(* CODESYS project Library01.library
   Company: MyCompany
   DefaultNamespace: MyNamespace01
   Version: 2.0.0.0
   Placeholder: MyLibrary01
   Title: MyLibrary01

Project tree, tasks and I/O mapping:
  libraries: Tc2_Standard, * (Beckhoff Automation GmbH); Tc2_System, * (Beckhoff Automation GmbH); Tc3_Module, * (Beckhoff Automation GmbH)
  DUTs/
    data type E_Foo
    data type ST_Foo
  GVLs/
    global variables GVL01
  POUs/
    function block FB_Foo [ST]
    interface I_Foo: DoSomething
  Version/
    global variables Global_Version
  VISUs/
*)

// DUTs/E_Foo
// {attribute 'qualified_only'}
// {attribute 'strict'}
TYPE E_Foo :
(
	eRed := 0,
	eBlue := 1,
	eGreen := 2
);
END_TYPE

// DUTs/ST_Foo
TYPE ST_Foo :
STRUCT
	bVal01	:	BOOL;
	bVal02	:	BOOL;
END_STRUCT
END_TYPE

// GVLs/GVL01
VAR_GLOBAL
	var01		:	INT;
END_VAR

// Version/Global_Version
{attribute 'TcGenerated'}
// This function has been automatically generated from the project information.
VAR_GLOBAL CONSTANT
	{attribute 'const_non_replaced'}
	{attribute 'linkalways'}
	stLibVersion_MyLibrary01 : ST_LibVersion := (iMajor := 2, iMinor := 0, iBuild := 0, iRevision := 0, sVersion := '2.0.0.0');
END_VAR

// POUs/FB_Foo
FUNCTION_BLOCK PUBLIC FB_Foo
VAR_INPUT
END_VAR
VAR_OUTPUT
END_VAR
VAR
END_VAR

END_FUNCTION_BLOCK

// POUs/I_Foo
INTERFACE I_Foo

METHOD DoSomething : BOOL
VAR_INPUT
END_VAR
END_METHOD

END_INTERFACE
